// SIMATIC S7-200 SMART project (STEP 7-Micro/WIN SMART), CPU SR20

SYMBOL_TABLE 系统符号
Clock_1s         SM0.5    // 针对 1 s 的周期时间，时钟脉冲接通 0.5 s，断开 0.5 s.
END_SYMBOL_TABLE

ORGANIZATION_BLOCK MAIN:OB1
TITLE=程序注释
BEGIN
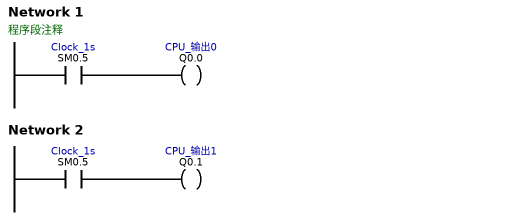
Network 1
// 程序段注释
LD     Clock_1s:SM0.5
=      CPU_输出0:Q0.0
Network 2
// (network saved uncompiled; LAD cells follow)
// row 0: c0 -| |- Clock_1s:SM0.5  c1 -( ) CPU_输出1:Q0.1
END_ORGANIZATION_BLOCK
